// TwinCAT 3 PLC project RT1
// ProgramVersion: 3.1.4026.17
// CompilerDefines: VISU_USEPROPERTYINFO
// libraries:
//   Tc2_Standard, * (Beckhoff Automation GmbH)
//   Tc2_System, * (Beckhoff Automation GmbH)
// project tree:
//   DUTs/ ST_EL8DO.TcDUT, st_OutputNums.TcDUT
//   / GlobalTextList.TcGTLO, PlcTask.TcTTO, Visualization Manager.TcVMO (not stored)
//   GVLs/ GVL_IO.TcGVL
//   POUs/ FB_EL8DO.TcPOU, MAIN.TcPOU
//   VISUs/ tl_OutputNames.TcTLO, Visualization.TcVIS
// real-time tasks:
//   TASK PlcTask: cycle T#10ms, priority 20, ADS port 350
// I/O:
//   DEVICE Device 1 (EtherCAT), AmsNetId 172.16.17.21.2.1
//     Term 1 (EK1200) [EK1200-5000 EtherCAT Power supply (2A E-Bus)]
//       Term 2 (EL2008) [EL2008 8Ch. Dig. Output 24V, 0.5A]
//       Term 3 (EK1322) [EK1322 2-port EtherCAT P junction with feed-in]
//       Term 4 (EL9011) [EL9011 End Terminal]
// variable links:
//   RT1/RT1 Instance <-> Device 1 (EtherCAT)/Term 1 (EK1200)/Term 2 (EL2008)
//     PlcTask Outputs/MAIN.el2008.digOutputs/do{1..8} <-> Channel {1..8}/Output  (8 links)

CONFIGURATION RT1
    RESOURCE PLC ON TwinCAT3
        TASK PlcTask(INTERVAL := T#10ms, PRIORITY := 20);
        PROGRAM MAIN WITH PlcTask : MAIN;
    END_RESOURCE
END_CONFIGURATION

// ---- DUTs/ST_EL8DO.TcDUT
TYPE ST_EL8DO :
STRUCT
	do1,do2,do3,do4,do5,do6,do7,do8:BOOL;
END_STRUCT
END_TYPE

// ---- DUTs/st_OutputNums.TcDUT
TYPE st_OutputNums :
STRUCT
	out1:		INT:=1;
	out2:		INT:=2;
	out3:		INT:=3;
	out4:       INT:=4;
	out5:       INT:=5;
	out6:       INT:=6;
	out7:       INT:=7;
	out8:       INT:=8;
END_STRUCT
END_TYPE

// ---- GVLs/GVL_IO.TcGVL
{attribute 'qualified_only'}
VAR_GLOBAL
	
END_VAR

// ---- POUs/MAIN.TcPOU
PROGRAM MAIN
VAR
	el2008: FB_EL8DO;
	outRefs: st_OutputNums;
	outs: ARRAY [1..8] OF BOOL;
END_VAR

el2008(outputRef:= outRefs, outputs:=outs );

END_PROGRAM

// ---- POUs/FB_EL8DO.TcPOU
FUNCTION_BLOCK FB_EL8DO
VAR_INPUT
	outputRef: st_OutputNums;
	outputs: ARRAY[1..8]OF BOOL;
END_VAR
VAR_OUTPUT
END_VAR
VAR
	digOutputs AT %Q*:ST_EL8DO;
	isValidConfig: BOOL;
END_VAR


IF isValidConfig THEN
	digOutputs.do1:=outputs[outputRef.out1];
	digOutputs.do2:=outputs[outputRef.out2];
	digOutputs.do3:=outputs[outputRef.out3];
	digOutputs.do4:=outputs[outputRef.out4];
	digOutputs.do5:=outputs[outputRef.out5];
	digOutputs.do6:=outputs[outputRef.out6];
	digOutputs.do7:=outputs[outputRef.out7];
	digOutputs.do8:=outputs[outputRef.out8];
END_IF

END_FUNCTION_BLOCK

// ---- VISUs/tl_OutputNames.TcTLO
TEXTLIST tl_OutputNames
  1 = 'Saida 01'
  2 = 'Saida 02'
  3 = 'Saida 03'
  4 = 'Saida 04'
  5 = 'Saida 05'
  6 = 'Saida 06'
  7 = 'Saida 07'
  8 = 'Saida 08'
   = ''
END_TEXTLIST

// ---- VISUs/Visualization.TcVIS
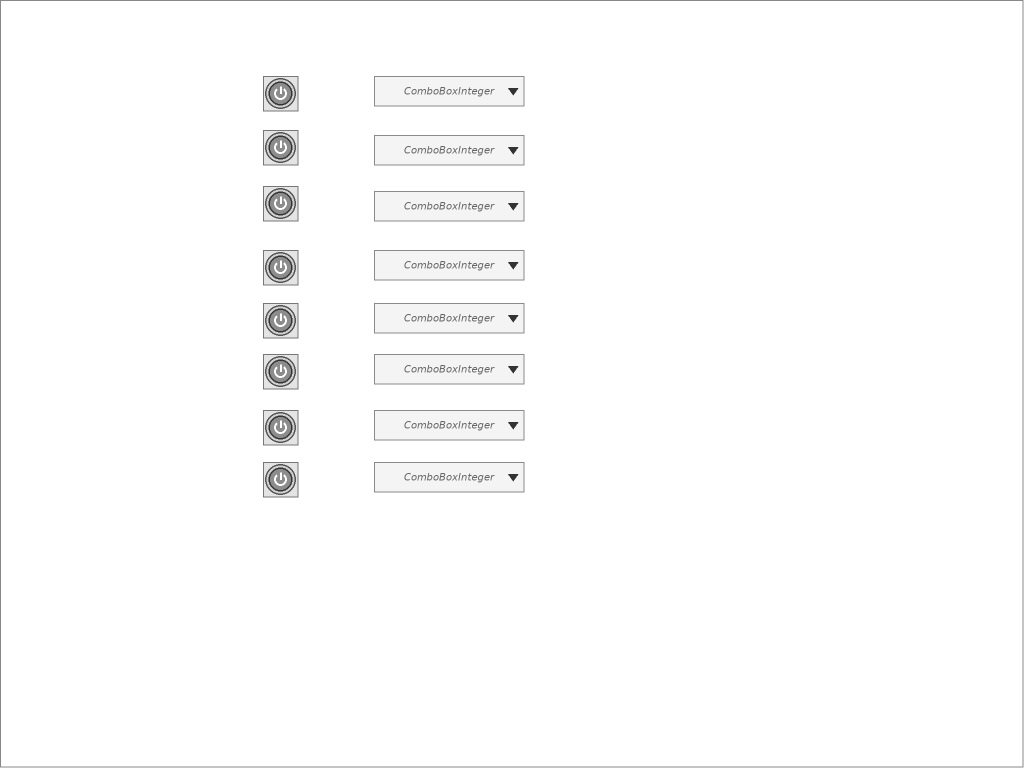
VISUALIZATION Visualization  // 1024x768
    ComboBoxInteger (374,76 150x30), variable: MAIN.outRefs.out1, text list: 'tl_OutputNames'
    ComboBoxInteger (374,135 150x30), variable: MAIN.outRefs.out2, text list: 'tl_OutputNames'
    ComboBoxInteger (374,191 150x30), variable: MAIN.outRefs.out3, text list: 'tl_OutputNames'
    ComboBoxInteger (374,250 150x30), variable: MAIN.outRefs.out4, text list: 'tl_OutputNames'
    ComboBoxInteger (374,303 150x30), variable: MAIN.outRefs.out5, text list: 'tl_OutputNames'
    ComboBoxInteger (374,354 150x30), variable: MAIN.outRefs.out6, text list: 'tl_OutputNames'
    ComboBoxInteger (374,410 150x30), variable: MAIN.outRefs.out7, text list: 'tl_OutputNames'
    ComboBoxInteger (374,462 150x30), variable: MAIN.outRefs.out8, text list: 'tl_OutputNames'
    PowerSwitch (263,76 35x35), variable: MAIN.outs[1], behaviour: TAP, style: Switch-PowerSwitch-Gray
    PowerSwitch (263,130 35x35), variable: MAIN.outs[2], behaviour: TAP, style: Switch-PowerSwitch-Gray
    PowerSwitch (263,186 35x35), variable: MAIN.outs[3], behaviour: TAP, style: Switch-PowerSwitch-Gray
    PowerSwitch (263,250 35x35), variable: MAIN.outs[4], behaviour: TAP, style: Switch-PowerSwitch-Gray
    PowerSwitch (263,303 35x35), variable: MAIN.outs[5], behaviour: TAP, style: Switch-PowerSwitch-Gray
    PowerSwitch (263,354 35x35), variable: MAIN.outs[6], behaviour: TAP, style: Switch-PowerSwitch-Gray
    PowerSwitch (263,410 35x35), variable: MAIN.outs[7], behaviour: TAP, style: Switch-PowerSwitch-Gray
    PowerSwitch (263,462 35x35), variable: MAIN.outs[8], behaviour: TAP, style: Switch-PowerSwitch-Gray
END_VISUALIZATION
